FUNCTION_BLOCK InfoDataAds EXTENDS InfoDataBase
VAR
	_AdsAddr AT %I*: AMSADDR;
END_VAR

PROPERTY AdsAddr : AMSADDR
GET
AdsAddr := _AdsAddr;
END_GET
END_PROPERTY

END_FUNCTION_BLOCK

(* stored: Version 1.1.0.1, ProductVersion 3.1.4024.9
   POU InfoDataAds: Id {ec4a6d3d-4b45-019c-1d05-3316b37b59d8}, SpecialFunc None
   Property AdsAddr: Id {0bfdfd08-9d77-0052-3a06-288bbd699273}
   Get Get: Id {57c95e47-3d0d-0c7d-2a8d-3493538a644c} *)
